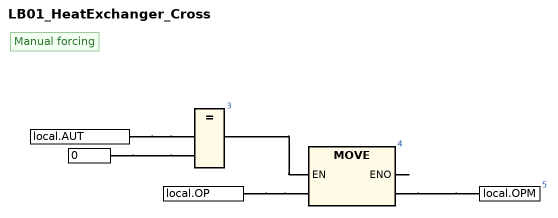
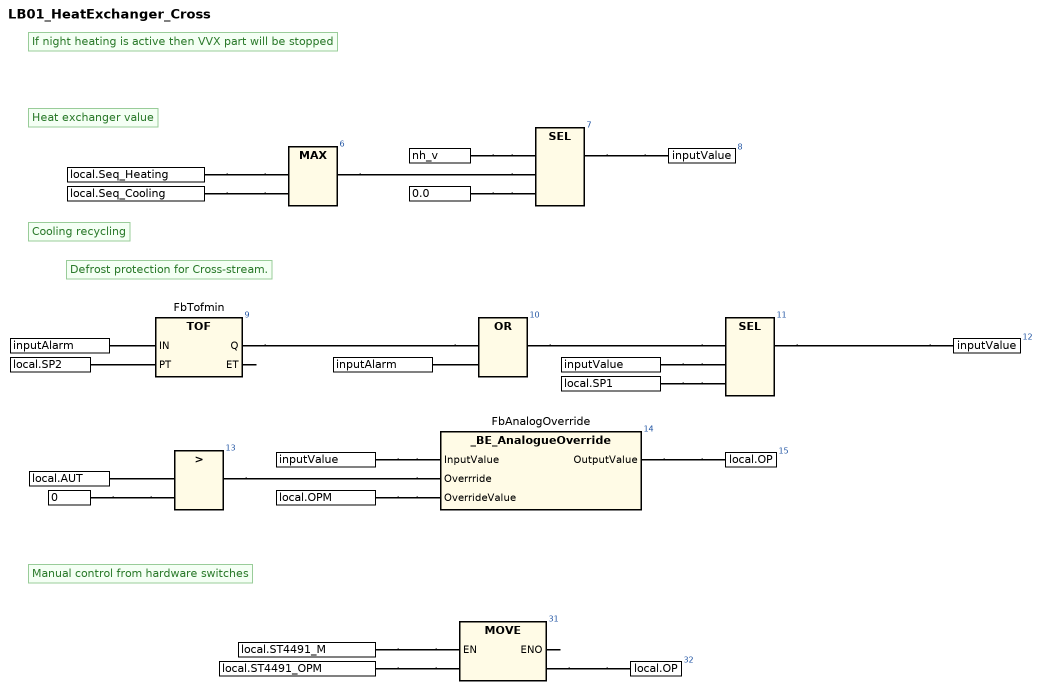
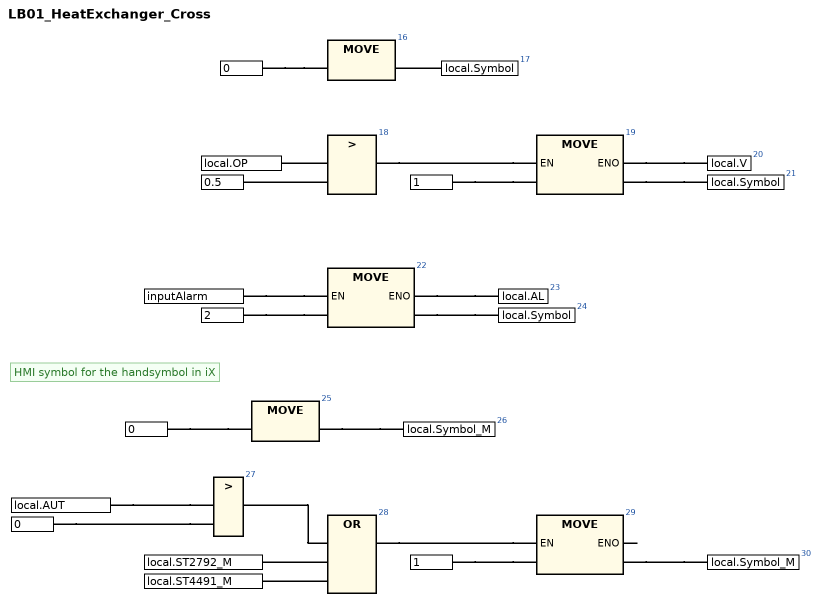
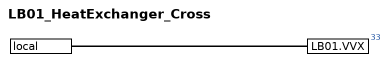
local := LB01.VVX;
inputAlarm := LB01.GP91.InputAlarm;
nh_v := LB01.NH.V;
// Manual forcing
IF local.AUT = 0 THEN _w1 := local.OP; END_IF
local.OPM := _w1;
// If night heating is active then VVX part will be stopped
// Heat exchanger value
inputValue := SEL(nh_v, MAX(local.Seq_Heating, local.Seq_Cooling), 0.0);
// Cooling recycling
// Defrost protection for Cross-stream.
FbTofmin(IN := inputAlarm, PT := local.SP2); // TOF
inputValue := SEL(FbTofmin.Q OR inputAlarm, inputValue, local.SP1);
FbAnalogOverride(InputValue := inputValue, Overrride := local.AUT > 0, OverrideValue := local.OPM); // _BE_AnalogueOverride
local.OP := FbAnalogOverride.OutputValue;
local.Symbol := 0;
_w2 := local.OP > 0.5;
IF _w2 THEN _w3 := 1; END_IF
local.V := _w2;
local.Symbol := _w3;
_w4 := inputAlarm;
IF _w4 THEN _w5 := 2; END_IF
local.AL := _w4;
local.Symbol := _w5;
// HMI symbol for the handsymbol in iX
local.Symbol_M := 0;
IF local.AUT > 0 OR local.ST2792_M OR local.ST4491_M THEN _w6 := 1; END_IF
local.Symbol_M := _w6;
// Manual control from hardware switches
IF local.ST4491_M THEN _w7 := local.ST4491_OPM; END_IF
local.OP := _w7;
LB01.VVX := local;

END_PROGRAM

// Device/AREA1/B001/LB01/Valve/SV91/LB01_SV91
PROGRAM LB01_SV91
VAR
	local:strValve;
	localGT:strSensor8_DefrostProt;
	FbAnalogueValve: _BE_AnalogueValve;
	fbExercise: _BE_Exercise;
	analogValue: REAL;
	valueFreezeProtection: REAL;
	FbAnalogOverride: _BE_AnalogueOverride;
	seqOutput: REAL;
	seqHeating: REAL;
	seqCooling: REAL;
	nh_v: BOOL;
	inputValue: REAL;
END_VAR
VAR // added by the converter: edge detectors and wires of the graphical bodies
    _w1, _w2, _w3, _w4 : ANY;
END_VAR

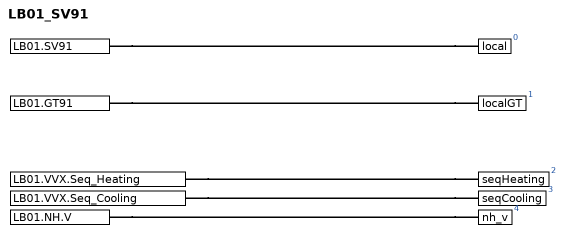
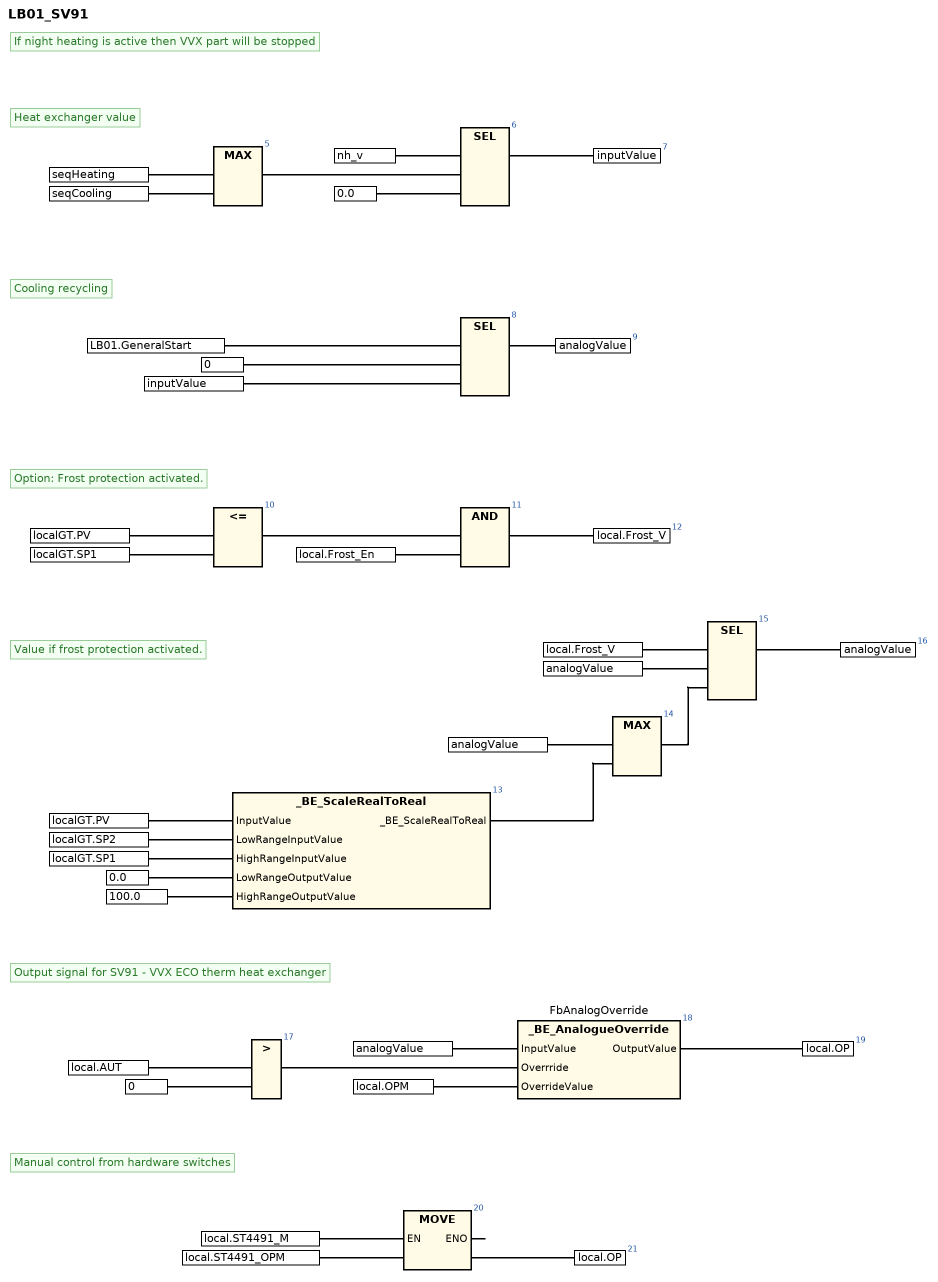
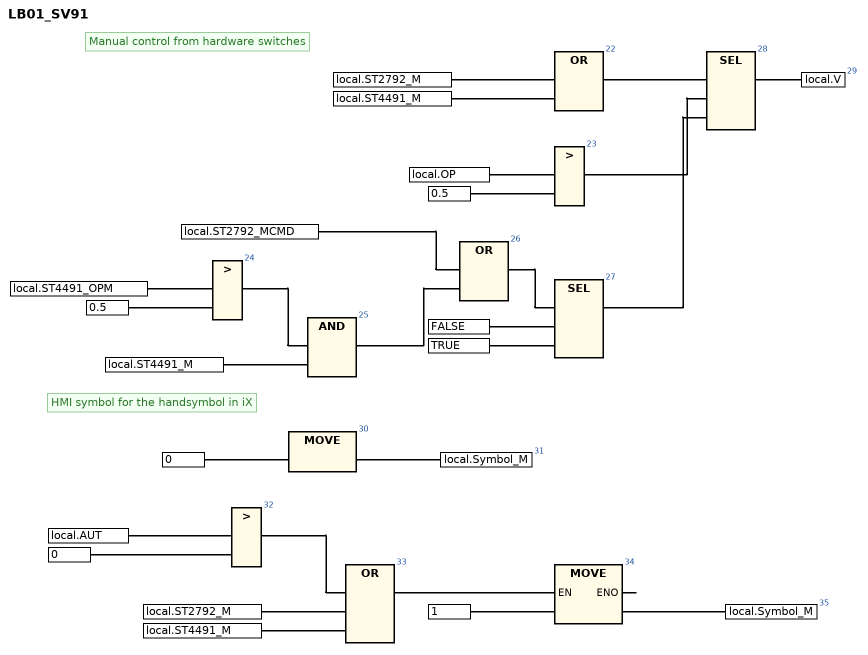
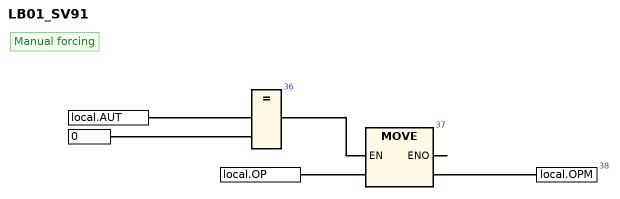
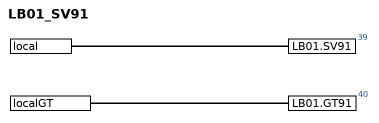
local := LB01.SV91;
localGT := LB01.GT91;
seqHeating := LB01.VVX.Seq_Heating;
seqCooling := LB01.VVX.Seq_Cooling;
nh_v := LB01.NH.V;
// If night heating is active then VVX part will be stopped
// Heat exchanger value
inputValue := SEL(nh_v, MAX(seqHeating, seqCooling), 0.0);
// Cooling recycling
analogValue := SEL(LB01.GeneralStart, 0, inputValue);
// Option: Frost protection activated.
local.Frost_V := localGT.PV <= localGT.SP1 AND local.Frost_En;
// Value if frost protection activated.
_w1 := _BE_ScaleRealToReal(InputValue := localGT.PV, LowRangeInputValue := localGT.SP2, HighRangeInputValue := localGT.SP1, LowRangeOutputValue := 0.0, HighRangeOutputValue := 100.0);
analogValue := SEL(local.Frost_V, analogValue, MAX(analogValue, _w1));
// Output signal for SV91 - VVX ECO therm heat exchanger
FbAnalogOverride(InputValue := analogValue, Overrride := local.AUT > 0, OverrideValue := local.OPM); // _BE_AnalogueOverride
local.OP := FbAnalogOverride.OutputValue;
// Manual control from hardware switches
IF local.ST4491_M THEN _w2 := local.ST4491_OPM; END_IF
local.OP := _w2;
// Manual control from hardware switches
local.V := SEL(local.ST2792_M OR local.ST4491_M, local.OP > 0.5, SEL(local.ST2792_MCMD OR local.ST4491_OPM > 0.5 AND local.ST4491_M, FALSE, TRUE));
// HMI symbol for the handsymbol in iX
local.Symbol_M := 0;
IF local.AUT > 0 OR local.ST2792_M OR local.ST4491_M THEN _w3 := 1; END_IF
local.Symbol_M := _w3;
// Manual forcing
IF local.AUT = 0 THEN _w4 := local.OP; END_IF
local.OPM := _w4;
LB01.SV91 := local;
LB01.GT91 := localGT;

END_PROGRAM

// Device/AREA1/B001/LB01/Pump/P3/LB01_P3
PROGRAM LB01_P3
VAR
	local:strPumpExercise;
	fbControlPump2: _BE_Pump_2;
	fbPumpStartCondition: _BE_PumpStartConditions;
	fb_OperationalTime: _BE_OperationalTime;
	fbExercise: _BE_Exercise;
	ackAl01: BOOL;
	ackAl02: BOOL;
	sv_op: REAL;
	startPump: BOOL;
	AlarmFbAL01: _BE_AlarmAckRequired;
	AlarmFbAL02: _BE_AlarmAckRequired;
END_VAR
VAR // added by the converter: edge detectors and wires of the graphical bodies
    _w1 : ANY;
END_VAR

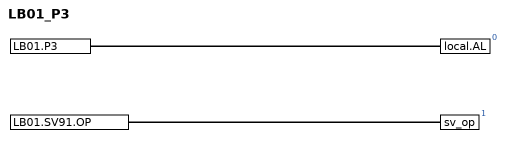
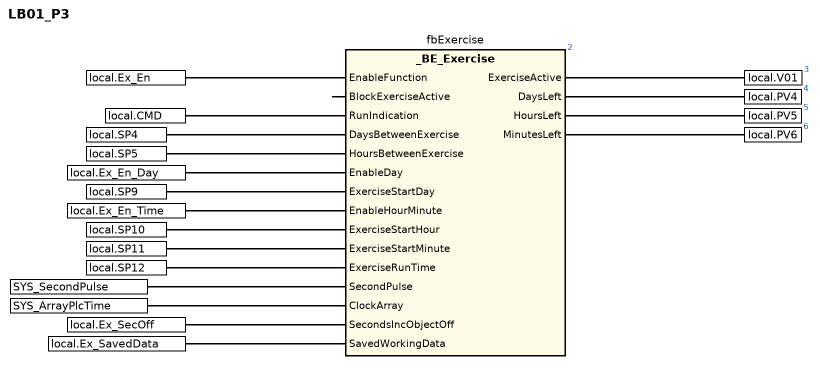
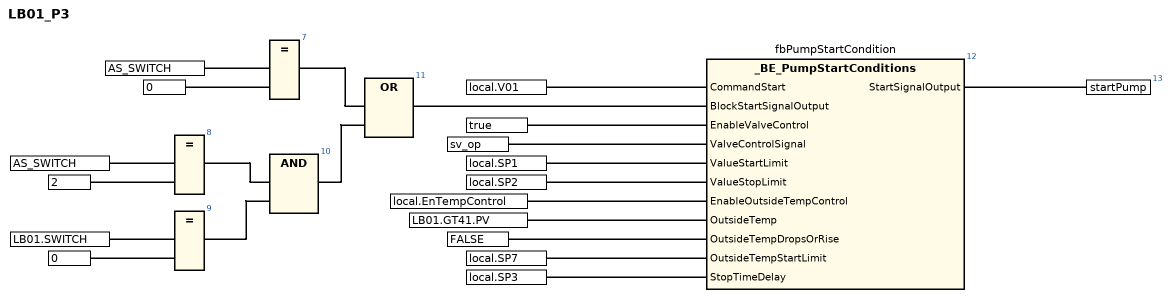
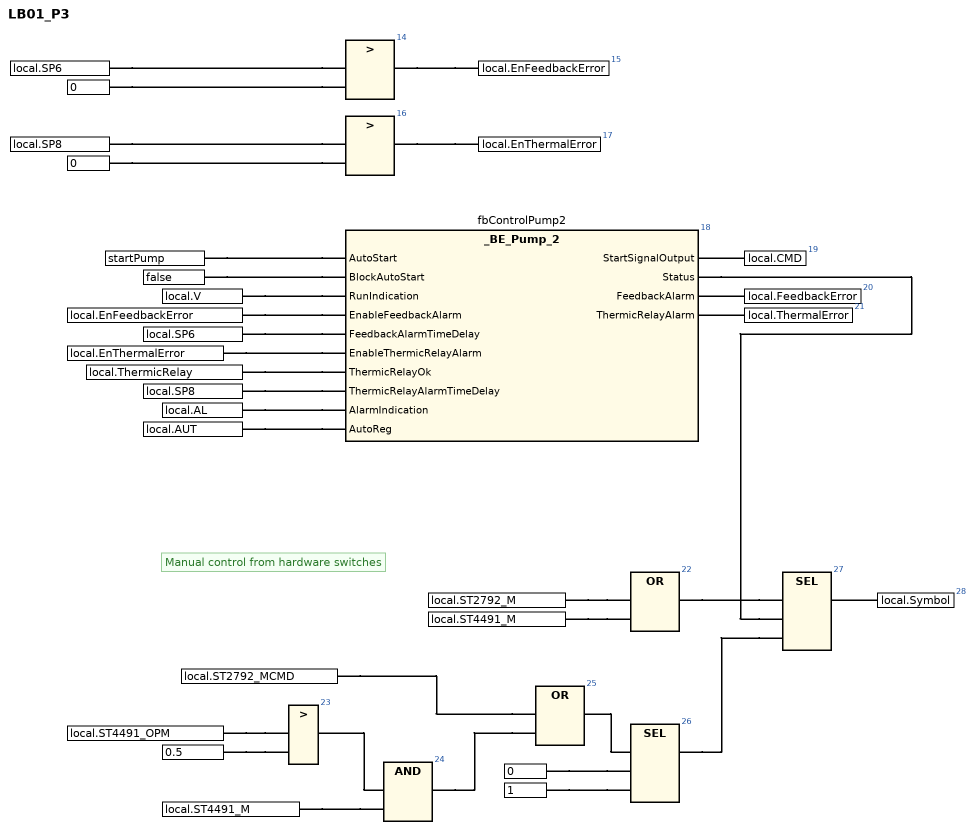
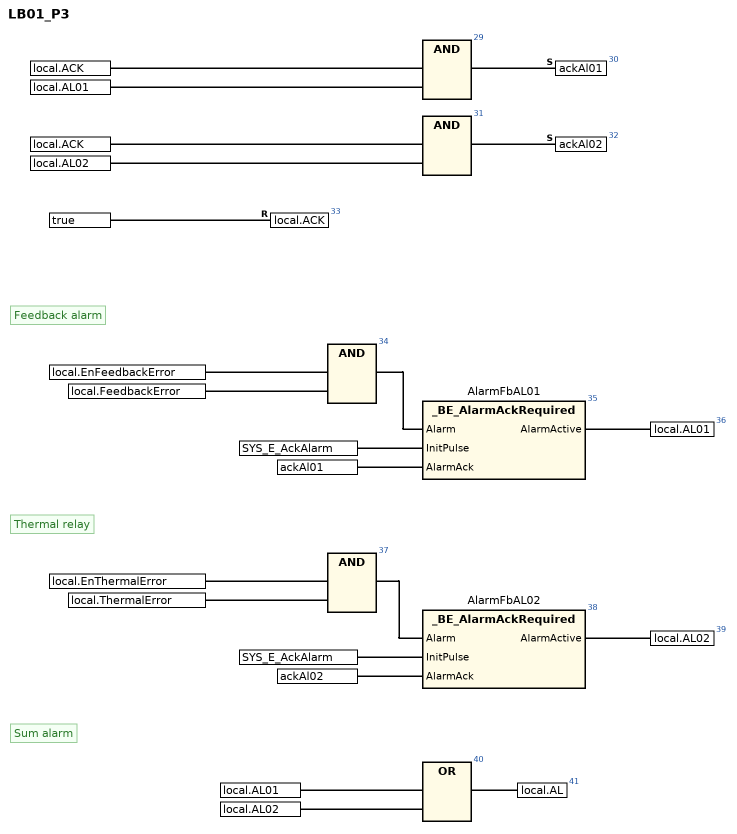
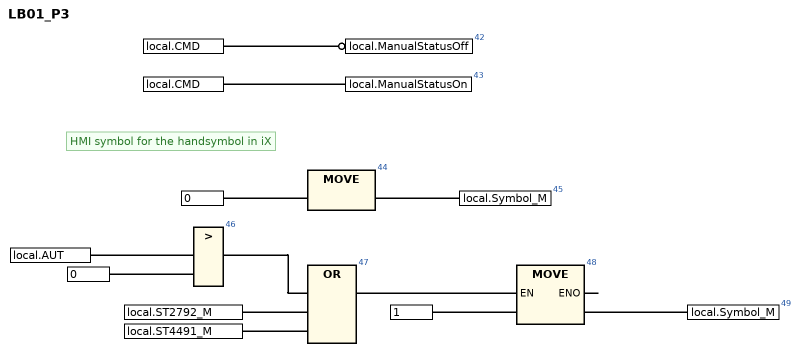
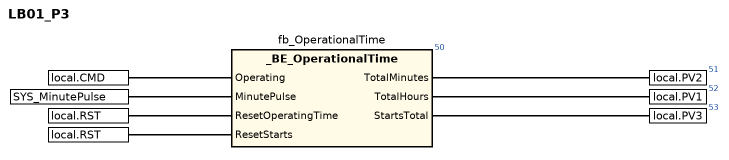
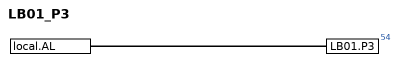
local.AL := LB01.P3;
sv_op := LB01.SV91.OP;
fbExercise(
    EnableFunction := local.Ex_En,
    RunIndication := local.CMD,
    DaysBetweenExercise := local.SP4,
    HoursBetweenExercise := local.SP5,
    EnableDay := local.Ex_En_Day,
    ExerciseStartDay := local.SP9,
    EnableHourMinute := local.Ex_En_Time,
    ExerciseStartHour := local.SP10,
    ExerciseStartMinute := local.SP11,
    ExerciseRunTime := local.SP12,
    SecondPulse := SYS_SecondPulse,
    ClockArray := SYS_ArrayPlcTime,
    SecondsIncObjectOff := local.Ex_SecOff,
    SavedWorkingData := local.Ex_SavedData); // _BE_Exercise
local.V01 := fbExercise.ExerciseActive;
local.PV4 := fbExercise.DaysLeft;
local.PV5 := fbExercise.HoursLeft;
local.PV6 := fbExercise.MinutesLeft;
fbPumpStartCondition(
    CommandStart := local.V01,
    BlockStartSignalOutput := AS_SWITCH = 0 OR AS_SWITCH = 2 AND LB01.SWITCH = 0,
    EnableValveControl := true,
    ValveControlSignal := sv_op,
    ValueStartLimit := local.SP1,
    ValueStopLimit := local.SP2,
    EnableOutsideTempControl := local.EnTempControl,
    OutsideTemp := LB01.GT41.PV,
    OutsideTempDropsOrRise := FALSE,
    OutsideTempStartLimit := local.SP7,
    StopTimeDelay := local.SP3); // _BE_PumpStartConditions
startPump := fbPumpStartCondition.StartSignalOutput;
local.EnFeedbackError := local.SP6 > 0;
local.EnThermalError := local.SP8 > 0;
fbControlPump2(
    AutoStart := startPump,
    BlockAutoStart := false,
    RunIndication := local.V,
    EnableFeedbackAlarm := local.EnFeedbackError,
    FeedbackAlarmTimeDelay := local.SP6,
    EnableThermicRelayAlarm := local.EnThermalError,
    ThermicRelayOk := local.ThermicRelay,
    ThermicRelayAlarmTimeDelay := local.SP8,
    AlarmIndication := local.AL,
    AutoReg := local.AUT); // _BE_Pump_2
local.CMD := fbControlPump2.StartSignalOutput;
local.FeedbackError := fbControlPump2.FeedbackAlarm;
local.ThermalError := fbControlPump2.ThermicRelayAlarm;
// Manual control from hardware switches
local.Symbol := SEL(local.ST2792_M OR local.ST4491_M, fbControlPump2.Status, SEL(local.ST2792_MCMD OR local.ST4491_OPM > 0.5 AND local.ST4491_M, 0, 1));
ackAl01 S= local.ACK AND local.AL01;
ackAl02 S= local.ACK AND local.AL02;
local.ACK R= true;
// Feedback alarm
AlarmFbAL01(
    Alarm := local.EnFeedbackError AND local.FeedbackError,
    InitPulse := SYS_E_AckAlarm,
    AlarmAck := ackAl01); // _BE_AlarmAckRequired
local.AL01 := AlarmFbAL01.AlarmActive;
// Thermal relay
AlarmFbAL02(
    Alarm := local.EnThermalError AND local.ThermalError,
    InitPulse := SYS_E_AckAlarm,
    AlarmAck := ackAl02); // _BE_AlarmAckRequired
local.AL02 := AlarmFbAL02.AlarmActive;
// Sum alarm
local.AL := local.AL01 OR local.AL02;
local.ManualStatusOff := NOT local.CMD;
local.ManualStatusOn := local.CMD;
// HMI symbol for the handsymbol in iX
local.Symbol_M := 0;
IF local.AUT > 0 OR local.ST2792_M OR local.ST4491_M THEN _w1 := 1; END_IF
local.Symbol_M := _w1;
fb_OperationalTime(
    Operating := local.CMD,
    MinutePulse := SYS_MinutePulse,
    ResetOperatingTime := local.RST,
    ResetStarts := local.RST); // _BE_OperationalTime
local.PV2 := fb_OperationalTime.TotalMinutes;
local.PV1 := fb_OperationalTime.TotalHours;
local.PV3 := fb_OperationalTime.StartsTotal;
LB01.P3 := local.AL;

END_PROGRAM

// Device/AREA1/B001/LB01/Sensor/Temperature/GT91/LB01_GT91
PROGRAM LB01_GT91
VAR
	local:strSensor8_DefrostProt;
	svOp: REAL;
	svFrost_V: BOOL;
	timerDefrost: TON;
	ackFault: BOOL;
	ackLal: BOOL;
	ackHal: BOOL;
	ackAl01: BOOL;
	gt_Min: TON;
	gt_Max: TON;
	AlarmAcknowledge01: _BE_AlarmAckRemote;
	AlarmAcknowledge02: _BE_AlarmAckRemote;
	AlarmAcknowledge03: _BE_AlarmAckRemote;
	AlarmAcknowledge04: _BE_AlarmAckRemote;
END_VAR
VAR // added by the converter: edge detectors and wires of the graphical bodies
    _w1, _w3, _w4 : ANY;
    _w2 : BOOL;
END_VAR

// note: 4 stored wires end on pins the file does not list and are not shown
local := LB01.GT91;
svOp := LB01.SV91.OP;
svFrost_V := LB01.SV91.Frost_V;
ackFault S= local.ACK AND local.FAULT;
ackLal S= local.ACK AND local.LAL;
ackHal S= local.ACK AND local.HAL;
ackAl01 S= local.ACK AND local.AL01;
local.ACK R= true;
// Sensor error
AlarmAcknowledge01(
    Alarm := local.PV < -3200.0 AND NOT SYS_StartupDelayComm,
    InitPulse := SYS_InitPulse,
    AlarmAck := ackFault); // _BE_AlarmAckRemote
local.FAULT := AlarmAcknowledge01.AlarmActive;
// Alarm Low
gt_Min(IN := local.PV < local.ALL AND NOT SYS_StartupDelayComm AND LB01.GeneralStart AND NOT local.FAULT, PT := DINT_TO_TIME(local.AD * 60000)); // TON
AlarmAcknowledge02(Alarm := gt_Min.Q, InitPulse := SYS_InitPulse, AlarmAck := ackLal); // _BE_AlarmAckRemote
local.LAL := AlarmAcknowledge02.AlarmActive;
// Alarm High
gt_Max(IN := local.PV > local.AHL AND NOT SYS_StartupDelayComm AND LB01.GeneralStart AND NOT local.FAULT, PT := DINT_TO_TIME(local.AD * 60000)); // TON
AlarmAcknowledge03(Alarm := gt_Max.Q, InitPulse := SYS_InitPulse, AlarmAck := ackHal); // _BE_AlarmAckRemote
local.HAL := AlarmAcknowledge03.AlarmActive;
// Defrost activated
timerDefrost(IN := svOp = 0.0 AND svFrost_V, PT := DINT_TO_TIME(local.AD1 * 60000)); // TON
AlarmAcknowledge04(Alarm := timerDefrost.Q, InitPulse := SYS_InitPulse, AlarmAck := ackAl01); // _BE_AlarmAckRemote
local.AL01 := AlarmAcknowledge04.AlarmActive;
// Status HMI
IF true THEN _w1 := 0; END_IF
local.Symbol := _w1;
_w2 := local.FAULT OR local.LAL OR local.HAL;
IF _w2 THEN _w3 := 2; END_IF
local.AL := _w2;
local.Symbol := _w3;
IF local.FAULT THEN _w4 := 3; END_IF
local.Symbol := _w4;
LB01.GT91 := local;
// al: input not connected

END_PROGRAM

// Device/AREA1/B001/LB01/Sensor/Pressure/GP61/LB01_GP61
PROGRAM LB01_GP61
VAR
	local:strSensor10_HeatExchanger_Pressure;
	AlarmAcknowledge01: _BE_AlarmAckRemote;
END_VAR
VAR // added by the converter: edge detectors and wires of the graphical bodies
    _w1, _w3 : ANY;
    _w2 : BOOL;
END_VAR

local := LB01.GP61;
// Alarm High
AlarmAcknowledge01(Alarm := local.InputAlarm, InitPulse := SYS_InitPulse, AlarmAck := local.ACK); // _BE_AlarmAckRemote
local.HAL := AlarmAcknowledge01.AlarmActive;
// Status i HMI
IF true THEN _w1 := 0; END_IF
local.Symbol := _w1;
_w2 := false OR local.HAL;
IF _w2 THEN _w3 := 2; END_IF
local.AL := _w2;
local.Symbol := _w3;
LB01.GP61 := local;

END_PROGRAM

// Device/AREA1/B001/LB01/Sensor/Pressure/GP12/LB01_GP12
PROGRAM LB01_GP12
VAR
	local:strSensor11_DiffPressure;
	AlarmAcknowledge01: _BE_AlarmAckRemote;
	fanGuardError: BOOL;
	timerAlarm: TON;
END_VAR
VAR // added by the converter: edge detectors and wires of the graphical bodies
    _w1, _w3 : ANY;
    _w2 : BOOL;
END_VAR

local := LB01.GP12;
// High alarm
timerAlarm(IN := local.V, PT := DINT_TO_TIME(local.AD * 60000)); // TON
AlarmAcknowledge01(Alarm := timerAlarm.Q, InitPulse := SYS_InitPulse, AlarmAck := local.ACK); // _BE_AlarmAckRemote
local.HAL := AlarmAcknowledge01.AlarmActive;
// Status i HMI
IF true THEN _w1 := 0; END_IF
local.Symbol := _w1;
_w2 := false OR local.HAL;
IF _w2 THEN _w3 := 2; END_IF
local.AL := _w2;
local.Symbol := _w3;
LB01.GP12 := local;

END_PROGRAM

// Device/AREA1/B001/LB01/Sensor/Pressure/GP22/LB01_GP22
PROGRAM LB01_GP22
VAR
	local:strSensor11_DiffPressure;
	AlarmAcknowledge01: _BE_AlarmAckRemote;
	fanGuardError: BOOL;
	timerAlarm: TON;
END_VAR
VAR // added by the converter: edge detectors and wires of the graphical bodies
    _w1, _w3 : ANY;
    _w2 : BOOL;
END_VAR

local := LB01.GP22;
// High alarm
timerAlarm(IN := local.V, PT := DINT_TO_TIME(local.AD * 60000)); // TON
AlarmAcknowledge01(Alarm := timerAlarm.Q, InitPulse := SYS_InitPulse, AlarmAck := local.ACK); // _BE_AlarmAckRemote
local.HAL := AlarmAcknowledge01.AlarmActive;
// Status i HMI
IF true THEN _w1 := 0; END_IF
local.Symbol := _w1;
_w2 := false OR local.HAL;
IF _w2 THEN _w3 := 2; END_IF
local.AL := _w2;
local.Symbol := _w3;
LB01.GP22 := local;

END_PROGRAM

// Device/AREA1/B001/LB01/Sensor/Flow/GF11/LB01_GF11
PROGRAM LB01_GF11
VAR
	local:strSensor2_Regulator;
	gt_Min: TON;
	gt_Max: TON;
	reset_en: RS;
	ackLal: BOOL;
	ackHal: BOOL;
	AlarmAcknowledge01: _BE_AlarmAckRemote;
	AlarmAcknowledge02: _BE_AlarmAckRemote;
END_VAR
VAR // added by the converter: edge detectors and wires of the graphical bodies
    _w1, _w3 : ANY;
    _w2 : BOOL;
END_VAR

local := LB01.GF11;
ackLal S= local.ACK AND local.LAL;
ackHal S= local.ACK AND local.HAL;
local.ACK R= true;
// Alarm Low
local.CSP1 := local.SP - local.ADL;
gt_Min(IN := local.PV < local.CSP1 AND NOT SYS_StartupDelayComm AND LB01.GeneralStart AND LB01.TF1.Operating, PT := DINT_TO_TIME(local.AD * 60000)); // TON
AlarmAcknowledge01(Alarm := gt_Min.Q, InitPulse := SYS_InitPulse, AlarmAck := ackLal); // _BE_AlarmAckRemote
local.LAL := AlarmAcknowledge01.AlarmActive;
// Alarm High
local.CSP2 := local.SP + local.ADL;
gt_Max(IN := local.PV > local.CSP2 AND NOT SYS_StartupDelayComm AND LB01.GeneralStart AND LB01.TF1.Operating, PT := DINT_TO_TIME(local.AD * 60000)); // TON
AlarmAcknowledge02(Alarm := gt_Max.Q, InitPulse := SYS_InitPulse, AlarmAck := ackHal); // _BE_AlarmAckRemote
local.HAL := AlarmAcknowledge02.AlarmActive;
// Status HMI
IF true THEN _w1 := 0; END_IF
local.Symbol := _w1;
_w2 := local.LAL OR local.HAL;
IF _w2 THEN _w3 := 2; END_IF
local.AL := _w2;
local.Symbol := _w3;
LB01.GF11 := local;

END_PROGRAM

// Device/AREA1/B001/LB01/Sensor/Flow/GF21/LB01_GF21
PROGRAM LB01_GF21
VAR
	local:strSensor2_Regulator;
	gt_Min: TON;
	gt_Max: TON;
	reset_en: RS;
	ackLal: BOOL;
	ackHal: BOOL;
	AlarmAcknowledge01: _BE_AlarmAckRemote;
	AlarmAcknowledge02: _BE_AlarmAckRemote;
END_VAR
VAR // added by the converter: edge detectors and wires of the graphical bodies
    _w1, _w3 : ANY;
    _w2 : BOOL;
END_VAR

local := LB01.GF21;
ackLal S= local.ACK AND local.LAL;
ackHal S= local.ACK AND local.HAL;
local.ACK R= true;
// Alarm Low
local.CSP1 := local.SP - local.ADL;
gt_Min(IN := local.PV < local.CSP1 AND NOT SYS_StartupDelayComm AND LB01.GeneralStart AND LB01.TF1.Operating, PT := DINT_TO_TIME(local.AD * 60000)); // TON
AlarmAcknowledge01(Alarm := gt_Min.Q, InitPulse := SYS_InitPulse, AlarmAck := ackLal); // _BE_AlarmAckRemote
local.LAL := AlarmAcknowledge01.AlarmActive;
// Alarm High
local.CSP2 := local.SP + local.ADL;
gt_Max(IN := local.PV > local.CSP2 AND NOT SYS_StartupDelayComm AND LB01.GeneralStart AND LB01.TF1.Operating, PT := DINT_TO_TIME(local.AD * 60000)); // TON
AlarmAcknowledge02(Alarm := gt_Max.Q, InitPulse := SYS_InitPulse, AlarmAck := ackHal); // _BE_AlarmAckRemote
local.HAL := AlarmAcknowledge02.AlarmActive;
// Status HMI
IF true THEN _w1 := 0; END_IF
local.Symbol := _w1;
_w2 := local.LAL OR local.HAL;
IF _w2 THEN _w3 := 2; END_IF
local.AL := _w2;
local.Symbol := _w3;
LB01.GF21 := local;

END_PROGRAM

// Device/AREA1/B001/LB01/Function/LB01_Function_AirQuality
PROGRAM LB01_Function_AirQuality
VAR
	fb_airQuality: _BE_AirQuality;
	analogValueSvAQ: REAL;
	fb_analogOverrideST11: _BE_AnalogueOverride;
	fb_analogOverrideST21: _BE_AnalogueOverride;
	timerCo2: TON;
END_VAR

// Air Quality Control
fb_airQuality(
    Co2DetectorValue := LB01.GQ31.PV,
    Co2LowLimit := LB01.GQ31.LL,
    Co2HighLimit := LB01.GQ31.HL,
    OutputMin := LB01.GQ31.MIN1,
    OutputMax := LB01.GQ31.MAX1); // _BE_AirQuality
timerCo2(IN := fb_airQuality.Co2HighAlarm, PT := DINT_TO_TIME(LB01.GQ31.AD * 60000)); // TON
LB01.GQ31.HighAlarm := timerCo2.Q;
analogValueSvAQ := SEL(LB01.NC.V, SEL(LB01.GeneralStart, 0.0, fb_airQuality.OutputValue), 100.0);
// Output value for ST11
fb_analogOverrideST11(
    InputValue := analogValueSvAQ,
    Overrride := LB01.ST11.AUT > 0,
    OverrideValue := LB01.ST11.OPM); // _BE_AnalogueOverride
LB01.ST11.OP := fb_analogOverrideST11.OutputValue;
// Output value for ST21
fb_analogOverrideST21(
    InputValue := analogValueSvAQ,
    Overrride := LB01.ST21.AUT > 0,
    OverrideValue := LB01.ST21.OPM); // _BE_AnalogueOverride
LB01.ST21.OP := fb_analogOverrideST21.OutputValue;

END_PROGRAM

// Device/AREA1/B001/LB01/Fan/FF1/LB01_FF1_Analog_ST
PROGRAM LB01_FF1_Analog_ST
VAR
	local:strFan_Analog;
	localGP:strSensor2_Regulator;
	ControlFan: _BE_Fan;
	FbRegulator: _BE_Regulator;
	_BE_Fan2: _BE_Fan_2;
	reset_en: RS;
	AlarmFbAl03: _BE_AlarmAckRequired;
	AlarmFbAl02: _BE_AlarmAckRequired;
	fb_OperationalTime: _BE_OperationalTime;
	ackAl01: BOOL;
	ackAl02: BOOL;
	fanGuardOk: BOOL;
END_VAR

//Struct ->> local
LB01.FF1 := local;
LB01.GP21 := localGP;
LB01.GP23.V := fanGuardOk;

//Fan
IF Local.SP2 > 0 THEN
	local.EnFeedbackError := TRUE;
END_IF

IF Local.SP1 > 0 THEN
	local.EnThermalError := TRUE;
END_IF

IF Local.SP3 > 0 THEN
	local.EnFanGuardError := TRUE;
END_IF

_BE_Fan2.AutoStart := LB01.GeneralStart;
_BE_Fan2.AutoStartTimeDelay := local.SP1 + 5; 
_BE_Fan2.BlockAutoStart := FALSE;
_BE_Fan2.RunIndication := local.V; 
_BE_Fan2.EnableFeedbackAlarm := local.EnFeedbackError; 
_BE_Fan2.FeedbackAlarmTimeDelay := local.SP4; 
_BE_Fan2.EnableThermicRelayAlarm := local.EnThermalError;
_BE_Fan2.ThermicRelayOk := local.ThermoRelay1;
_BE_Fan2.ThermicRelayAlarmTimeDelay := local.SP2;
_BE_Fan2.EnableFanGuardAlarm := local.EnFanGuardError;
_BE_Fan2.FanGuardOk := fanGuardOk;
_BE_Fan2.FanGuardAlarmTimeDelay := local.SP3;
_BE_Fan2.AlarmIndication := local.AL;
_BE_Fan2.AutoReg := local.AUT;

_BE_Fan2();

local.CMD := _BE_Fan2.StartSignalOutput; 
// _BE_Fan2.Status 
local.FeedbackError := _BE_Fan2.FeedbackAlarm;
local.ThermalError := _BE_Fan2.ThermicRelayAlarm;
local.FanGuardError := _BE_Fan2.FanGuardAlarm;

 

//Alarm

//Regulator

//Operational time
fb_OperationalTime(Operating := local.CMD, MinutePulse := SYS_MinutePulse, ResetOperatingTime := local.RST, ResetStarts := local.RST);
local.PV2 := fb_OperationalTime.TotalMinutes;
local.PV1 := fb_OperationalTime.TotalHours;
local.PV3 := fb_OperationalTime.StartsTotal;

//Local --> STRUCT
local := LB01.FF1;
localGP := LB01.GP21;

END_PROGRAM

// Device/AREA1/Testing Center/Test
PROGRAM Test
VAR
	
END_VAR

//Indata to test loop
LB01.FF1.SP1 := 50;

//Evaluate result and report
IF LB01.FF1.RunIndication = TRUE THEN
	WriteLineInFile("c:Result", "2018-12-05 11:10:20 - FF1 - Running indicator working");
END_IF

END_PROGRAM

// Device/AREA1/B001/LB01/Fan/FF2/LB01_FF2_Analog_ST
PROGRAM LB01_FF2_Analog_ST
VAR
	local:strFan_Analog;
	localGP:strSensor2_Regulator;
	ControlFan: _BE_Fan;
	FbRegulator: _BE_Regulator;
	_BE_Fan2: _BE_Fan_2;
	reset_en: RS;
	AlarmFbAl03: _BE_AlarmAckRequired;
	AlarmFbAl02: _BE_AlarmAckRequired;
	fb_OperationalTime: _BE_OperationalTime;
	ackAl01: BOOL;
	ackAl02: BOOL;
	fanGuardOk: BOOL;
END_VAR

//Struct ->> local
LB01.FF2 := local;
LB01.GP21 := localGP;
LB01.GP23.V := fanGuardOk;

//Fan
IF Local.SP2 > 0 THEN
	local.EnFeedbackError := TRUE;
END_IF

IF Local.SP1 > 0 THEN
	local.EnThermalError := TRUE;
END_IF

IF Local.SP3 > 0 THEN
	local.EnFanGuardError := TRUE;
END_IF

_BE_Fan2.AutoStart := LB01.GeneralStart;
_BE_Fan2.AutoStartTimeDelay := local.SP1 + 5; 
_BE_Fan2.BlockAutoStart := FALSE;
_BE_Fan2.RunIndication := local.V; 
_BE_Fan2.EnableFeedbackAlarm := local.EnFeedbackError; 
_BE_Fan2.FeedbackAlarmTimeDelay := local.SP4; 
_BE_Fan2.EnableThermicRelayAlarm := local.EnThermalError;
_BE_Fan2.ThermicRelayOk := local.ThermoRelay1;
_BE_Fan2.ThermicRelayAlarmTimeDelay := local.SP2;
_BE_Fan2.EnableFanGuardAlarm := local.EnFanGuardError;
_BE_Fan2.FanGuardOk := fanGuardOk;
_BE_Fan2.FanGuardAlarmTimeDelay := local.SP3;
_BE_Fan2.AlarmIndication := local.AL;
_BE_Fan2.AutoReg := local.AUT;

_BE_Fan2();

local.CMD := _BE_Fan2.StartSignalOutput; 
// _BE_Fan2.Status 
local.FeedbackError := _BE_Fan2.FeedbackAlarm;
local.ThermalError := _BE_Fan2.ThermicRelayAlarm;
local.FanGuardError := _BE_Fan2.FanGuardAlarm;

 

//Alarm

//Regulator

//Operational time
fb_OperationalTime(Operating := local.CMD, MinutePulse := SYS_MinutePulse, ResetOperatingTime := local.RST, ResetStarts := local.RST);
local.PV2 := fb_OperationalTime.TotalMinutes;
local.PV1 := fb_OperationalTime.TotalHours;
local.PV3 := fb_OperationalTime.StartsTotal;

//Local --> STRUCT
local := LB01.FF2;
localGP := LB01.GP21;

END_PROGRAM
